PROGRAM MODE_SELECTION
VAR
		
END_VAR

// MODE FUNTIONAL BLOCK

FB_MODE_BLOCK(
	ModeWord:= MODE_WORD, 
	HomeConditionOK:= ALL_STN_IN_HOME, 
	OperationEnable:= SAFE_TO_WORK, 
	StartPB:= START_PB , 
	SafetyAndNOError:= , 
	ModeAck:=MODE_CHANGE_ACK, 
	HomingINProgress:= , 
	TempHomeOK:= , 
	ResetPB:= RESET_PB, 
	AutoSelected=> AUTO_SELECTED, 
	ManualSelected=> MANUAL_SELECTED, 
	StepSelected=> STEP_SELECTED, 
	ModeSelAck_Indication=> , 
	StatusDisplay=> , 
	AutoRunning:= AUTO_RUNNING, 
	StepRunning:= STEP_RUNNING, 
	StartEnable:= START_ENABLE, 
	MachineStop:= MACHINE_STOP);

END_PROGRAM

(* stored: Version 1.1.0.1, ProductVersion 3.1.4024.11
   POU MODE_SELECTION: Id {62466ff8-8bc6-4aa9-b792-aaf55af543d7}, SpecialFunc None *)
